# B&R Automation Studio project stroj
Automation Studio 4.10.2.37; technology packages: mapp 5.14.1, mappView 5.14.2

## Configuration Config1

CPU 4PPC30.0702-22B, AutomationRuntime B4.91, Build 4.1.2, Vc V4.72.3

CPU 4PPC30.0702-23B, AutomationRuntime B4.91, Build 4.1.2, Vc V4.72.3

### Task classes (Cpu.sw)
```
Cyclic#1 (cycle 10000 us, tolerance 10000 us):
  TempReg <- TempReg.prg
Cyclic#3 (cycle 50000 us, tolerance 50000 us):
  Machine_Co <- Machine_Control.prg
  Recipes <- Recipes.prg
  VizControl <- Visualization.VizControls.prg
VcDataObjects: Visu <- Visualization.Visu.dob
Binaries: mvLoader, FWRules, arsvcreg, udbdef, TCData, vcnet, vcrt, vccnum, vctcal, vcdsint, Visu03, vcfile, vcgclass, vccstr, vcpdsw, vccshape, arial, vccbmp, vcmgr, vcshared, vcdsloc, vcctext, Visu02, vccovl, vcfntttf, arialbd, vcalarm, vcpdvnc, vcpfar00, vccbtn, Visu01, vcbclass, vcclbox, arconfig, User, Role, Config, iomap, asfw, ashwac, ashwd, sysconf
Libraries: standard, MpRecipe, MpBase, sys_lib, runtime, MpFile, FileIO, astime, arssl, asieccon, vcresman, asbrstr, asusb, dataobj
```

### Task classes (Cpu.sw)
```
Cyclic#3 (cycle 50000 us, tolerance 50000 us):
  Machine_Co <- Machine_Control.prg
Cyclic#4 (cycle 100000 us, tolerance 100000 us):
  Recipes <- Recipes.prg
  VizControl <- VizControls.prg
VcDataObjects: Visu <- Visualization.Visu.dob
Binaries: mvLoader, FWRules, arsvcreg, udbdef, TCData, arconfig, User, Role, Config, iomap, asfw, ashwac, ashwd, sysconf
Libraries: standard, MpRecipe, MpBase, sys_lib, runtime, astime, arssl, asieccon, MpFile, FileIO
```

### Hardware
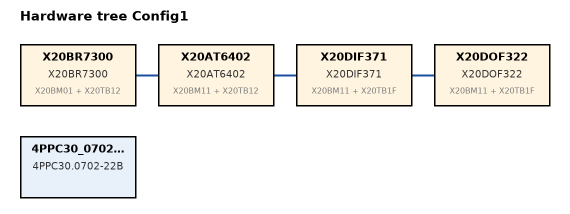
```
4PPC30_0702_22B : 4PPC30.0702-22B v1.1.3.0
  Connector IF3:
    ActivateDevice = 1
    Mode = Manual
    InternetAddress = 192.168.0.1
    SubnetMask = 255.255.255.0
    Vnc1
    VncKeyMappingFile1 = VC\PS2-Keyboard1.dis
    VncAuthentication1 = 1
    VncPasswordViewOnly1 = v
    VncPasswordViewControl1 = c
    VncMaxConnections1 = 4
    ActivateSnmp = 2
  Connector IF4:
    DeviceParam = /IF=2
    TerminatingResistor = 1
  Connector IF8:
    DeviceParam = /CLK=1843200 /CARD=68 /IF=1
  ConfigurationID = stroj_Config1
  EnableUsbRemoteInstall = 1
  TimerDeviceType = SWIOTIMER
  Cyclic1Duration = 10000
  Cyclic1Tolerance = 10000
  Cyclic2Duration = 20000
  Cyclic2Tolerance = 20000
  Cyclic3Duration = 50000
  Cyclic3Tolerance = 50000
  Cyclic4Duration = 100000
  Cyclic4Tolerance = 100000
  Cyclic5Duration = 200000
  Cyclic5Tolerance = 200000
  Cyclic6Duration = 500000
  Cyclic6Tolerance = 500000
  Cyclic7Duration = 1000000
  Cyclic7Tolerance = 1000000
  Cyclic8Duration = 10000
  Cyclic8Tolerance = 30000000
  FileDevice1
  FileDeviceName1 = Recipe
  FileDevicePath1 = C:\Projects\Recipes
  ActivateDtmServer = 1
  VcObjectName = Visu
  RotationAngle = 180
  KeyMappingFile = VC\4PPC30_0702_22B.dis
X20AT6402 : X20AT6402 v1.1.0.0  [SS1 -> X20TB12a.SS; SL -> X20BM11.SL1]
  FunctionModel = CANIOBusController
X20BM01 : X20BM01 v2.1.0.0
X20BM11 : X20BM11 v1.0.0.1  [X2X1 -> X20BM01.IF1]
X20BM11a : X20BM11 v1.0.0.1  [X2X1 -> X20BM11.X2X2]
X20BM11b : X20BM11 v1.0.0.1  [X2X1 -> X20BM11a.X2X2]
X20BR7300 : X20BR7300 v1.4.0.0  [CAN1 -> 4PPC30_0702_22B.IF4; SL -> X20BM01.SL1; SS1 -> X20TB12.SS]
  Supervision = off
X20DIF371 : X20DIF371 v1.1.0.0  [SS1 -> X20TB1F.SS; SL -> X20BM11a.SL1]
  FunctionModel = CANIOBusController
X20DOF322 : X20DOF322 v1.4.0.0  [SS1 -> X20TB1F1.SS; SL -> X20BM11b.SL1]
  FunctionModel = CANIOBusController
X20TB12 : X20TB12 v1.0.0.0
X20TB12a : X20TB12 v1.0.0.0
X20TB1F : X20TB1F v1.0.0.0
X20TB1F1 : X20TB1F v1.0.0.0
```

### IoMap.iom - 4PPC30_0702_23B/IoMap.iom
```iecst
VAR_CONFIG
	::gDoHeatingZone1 AT %QX."X20DOF322".DigitalOutput05; (*24 VDC / 0.5 A, source (Heat zone 1)*)
	::gDoHeatingZone2 AT %QX."X20DOF322".DigitalOutput07; (*24 VDC / 0.5 A, source (Heat zone 2)*)
	::gDoHeatingZone3 AT %QX."X20DOF322".DigitalOutput11; (*24 VDC / 0.5 A, source (Heat zone 3)*)
	::gCurrentTemperatures.temperatureHeatZone1 AT %IW."X20AT6402".Temperature01;
	::gCurrentTemperatures.temperatureHeatZone2 AT %IW."X20AT6402".Temperature02;
	::gCurrentTemperatures.temperatureHeatZone3 AT %IW."X20AT6402".Temperature03;
	::gCurrentTemperatures.temperatureIRSensor AT %IW."X20AT6402".Temperature05;
	::gDoVacuum AT %QX."X20DOF322".DigitalOutput02;
	::gDoFreeItem AT %QX."X20DOF322".DigitalOutput04;
	::gDoMaterial AT %QX."X20DOF322".DigitalOutput06;
	::gDoHeating AT %QX."X20DOF322".DigitalOutput08;
	::gDoFrameDown AT %QX."X20DOF322".DigitalOutput10;
	::gDoFrameUp AT %QX."X20DOF322".DigitalOutput12;
	::gDoFormUp AT %QX."X20DOF322".DigitalOutput14;
	::gDoLedControl AT %QX."X20DOF322".DigitalOutput15;
	::gDoCooling AT %QX."X20DOF322".DigitalOutput01;
	::gDoAirPump AT %QX."X20DOF322".DigitalOutput03;
	::gDiSafe_OK AT %IX."X20DIF371".DigitalInput01;
	::gDiQF1_OK AT %IX."X20DIF371".DigitalInput11;
	::gDiQF2_OK AT %IX."X20DIF371".DigitalInput13;
	::gDiQF3_OK AT %IX."X20DIF371".DigitalInput15;
	::gDiButtonStart AT %IX."X20DIF371".DigitalInput03;
	::gDiHeatingLow AT %IX."X20DIF371".DigitalInput02;
	::gDiHeatingHigh AT %IX."X20DIF371".DigitalInput04;
	::gDiFrameUpPoistion AT %IX."X20DIF371".DigitalInput06;
	::gDiFrameDownPosition AT %IX."X20DIF371".DigitalInput08;
	::gDiFormDownPosition AT %IX."X20DIF371".DigitalInput10;
	::gDiFormUpPosition AT %IX."X20DIF371".DigitalInput12;
END_VAR
```

## Configuration Final

CPU 4PPC30.0702-22B, AutomationRuntime B4.91, Build 4.1.2, Vc V4.72.3

### Task classes (Cpu.sw)
```
Cyclic#1 (cycle 10000 us, tolerance 10000 us):
  TempReg <- TempReg.prg
Cyclic#3 (cycle 50000 us, tolerance 50000 us):
  Machine_Co <- Machine_Control.prg
  Recipes <- Recipes.prg
  VizControl <- Visualization.VizControls.prg
VcDataObjects: Visu <- Visualization.Visu.dob
Binaries: udbdef, mvLoader, FWRules, TCData, sysconf, Role, User, iomap, ashwd, asfw, arconfig, ashwac
Libraries: runtime, arssl, fileio
```

### Hardware
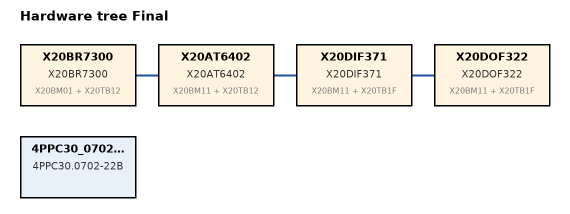
```
4PPC30_0702_22B : 4PPC30.0702-22B v1.1.3.0
  Connector IF3:
    ActivateDevice = 1
  ConfigurationID = stroj_Final
  Simulation = 1
  TimerDeviceType = SWIOTIMER
  Cyclic1Duration = 10000
  Cyclic1Tolerance = 10000
  Cyclic2Duration = 20000
  Cyclic2Tolerance = 20000
  Cyclic3Duration = 50000
  Cyclic3Tolerance = 50000
  Cyclic4Duration = 100000
  Cyclic4Tolerance = 100000
  Cyclic5Duration = 200000
  Cyclic5Tolerance = 200000
  Cyclic6Duration = 500000
  Cyclic6Tolerance = 500000
  Cyclic7Duration = 1000000
  Cyclic7Tolerance = 1000000
  Cyclic8Duration = 10000
  Cyclic8Tolerance = 30000000
  FileDevice1
  FileDeviceName1 = Recipes
  FileDevicePath1 = D:\
  VcObjectName = Visu
  RotationAngle = 180
  KeyMappingFile = VC\4PPC30_0702_22B.dis
X20AT6402 : X20AT6402 v1.1.0.0  [SS1 -> X20TB12.SS; SL -> X20BM11.SL1]
  FunctionModel = CANIOBusController
X20BM01a : X20BM01 v2.1.0.0
X20BM11 : X20BM11 v1.0.0.1  [X2X1 -> X20BM01a.IF1]
X20BM11a : X20BM11 v1.0.0.1  [X2X1 -> X20BM11.X2X2]
X20BM11b : X20BM11 v1.0.0.1  [X2X1 -> X20BM11a.X2X2]
X20BR7300 : X20BR7300 v1.4.0.0  [CAN1 -> 4PPC30_0702_22B.IF4 (NodeNumber=1); SL -> X20BM01a.SL1; SS1 -> X20TB12a.SS]
X20DIF371 : X20DIF371 v1.1.0.0  [SS1 -> X20TB1F.SS; SL -> X20BM11a.SL1]
  FunctionModel = CANIOBusController
X20DOF322 : X20DOF322 v1.4.0.0  [SS1 -> X20TB1F1.SS; SL -> X20BM11b.SL1]
  FunctionModel = CANIOBusController
X20TB12 : X20TB12 v1.0.0.0
X20TB12a : X20TB12 v1.0.0.0
X20TB1F : X20TB1F v1.0.0.0
X20TB1F1 : X20TB1F v1.0.0.0
```

### IoMap.iom - 4PPC30_0702_22B/IoMap.iom
```iecst
VAR_CONFIG
	::gDiSafe_OK AT %IX."X20DIF371".DigitalInput01;
	::gDiHeatingBack AT %IX."X20DIF371".DigitalInput02;
	::gDiQF1_OK AT %IX."X20DIF371".DigitalInput11 INVERSE;
	::gDiQF2_OK AT %IX."X20DIF371".DigitalInput13 INVERSE;
	::gDiQF3_OK AT %IX."X20DIF371".DigitalInput15 INVERSE;
	::gDiHeatingFront AT %IX."X20DIF371".DigitalInput04;
	::gDiFrameUpPoistion AT %IX."X20DIF371".DigitalInput06;
	::gDiFrameDownPosition AT %IX."X20DIF371".DigitalInput08;
	::gDiFormDownPosition AT %IX."X20DIF371".DigitalInput10;
	::gDiButtonStart AT %IX."X20DIF371".DigitalInput03;
	::gDoCooling AT %QX."X20DOF322".DigitalOutput01;
	::gDoHeatingZone1 AT %QX."X20DOF322".DigitalOutput05;
	::gDoHeatingZone2 AT %QX."X20DOF322".DigitalOutput07;
	::gDoLedControl AT %QX."X20DOF322".DigitalOutput15;
	::gDoVacuum AT %QX."X20DOF322".DigitalOutput02;
	::gDoAirPump AT %QX."X20DOF322".DigitalOutput03;
	::gDoFreeItem AT %QX."X20DOF322".DigitalOutput04;
	::gDoMaterial AT %QX."X20DOF322".DigitalOutput06;
	::gDoHeating AT %QX."X20DOF322".DigitalOutput08;
	::gDoFrameDown AT %QX."X20DOF322".DigitalOutput10;
	::gDoFrameUp AT %QX."X20DOF322".DigitalOutput12;
	::gDoFormUp AT %QX."X20DOF322".DigitalOutput14;
	::gCurrentTemperatures.temperatureHeatZone1 AT %IW."X20AT6402".Temperature01;
	::gCurrentTemperatures.temperatureHeatZone2 AT %IW."X20AT6402".Temperature02;
	::gCurrentTemperatures.temperatureHeatZone3 AT %IW."X20AT6402".Temperature03;
	::gCurrentTemperatures.temperatureIRSensor AT %IW."X20AT6402".Temperature05;
	::gDiFormUpPosition AT %IX."X20DIF371".DigitalInput12;
	::gDoHeatingZone3 AT %QX."X20DOF322".DigitalOutput09;
END_VAR
```

## Logical view

Binary libraries used (declarations not repeated): operator, runtime, astime, AsIecCon, standard, MpRecipe, MpBase, sys_lib

### Global.typ - Global data types
```iecst
TYPE
	StateOfProcessType :
		(
		ManualMode,
		DefaultState,
		Start,
		BubbleANDFormDownDelay,
		StartForming,
		CoolingANDBlowingDelay,
		Finishing
		);
	TemperaturesType : 	STRUCT
		temperatureHeatZone1 : INT;
		temperatureHeatZone2 : INT;
		temperatureHeatZone3 : INT;
		temperatureIRSensor : INT;
		temperatureOffset : INT;
		temperatureHysterese : REAL;
	END_STRUCT;
	TimersType : 	STRUCT
		HeatingTOFValue : REAL;
		BlowingTONValue : REAL;
		BlowingTOFValue : REAL;
		BubbleTOFValue : REAL;
		FormingTONValue : REAL;
		FormLockingTONValue : REAL;
		FormingTOFVALUE : REAL;
		FreeItemTOFValue : REAL;
		FreeItemTONValue : REAL;
		FormUpTONValue : REAL;
	END_STRUCT;
END_TYPE
```

### Global.var - Global variables
```iecst
VAR
	gDoMaterial : BOOL;
	gDiButtonStart : BOOL;
	gDiQF2_OK : BOOL;
	gDoCooling : BOOL;
	gDoAirPump : BOOL;
	gDiSafe_OK : BOOL;
	gDiQF1_OK : BOOL;
	gDiFrameUpPoistion : BOOL;
	gDiHeatingLow : BOOL;
	gDiHeatingHigh : BOOL;
	gDoFormUp : BOOL;
	gDiQF3_OK : BOOL;
	gDoLedControl : BOOL;
	gDoHeatingZone2 : BOOL;
	gDiFrameDownPosition : BOOL;
	gDoHeatingZone1 : BOOL;
	gDoVacuum : BOOL;
	gDoFreeItem : BOOL;
	gDoHeatingZone3 : BOOL;
	gDoFrameDown : BOOL;
	gDoFrameUp : BOOL;
	gDiFormDownPosition : BOOL;
	gDiFormUpPosition : BOOL;
	gDoHeating : BOOL;
	gAiIRSensor : INT;
	gAiHeatingZone1 : INT;
	gAiHeatingZone3 : INT;
	gAiHeatingZone2 : INT;
	gAVGTemperature : INT;
	gStateOfProcess : StateOfProcessType;
	gSetTemperatures : TemperaturesType;
	gSetTimersValues : TimersType;
	gRecipeLoaded : BOOL;
	gCurrentTemperatures : TemperaturesType;
	gDiHeatingFront : BOOL;
	gDiHeatingBack : BOOL;
	gHeatingZone1Ready : BOOL;
	gHeatingZone2Ready : BOOL;
	gHeatingZone3Ready : BOOL;
END_VAR
```


### Program Logical/Machine_Control (IEC)

#### Main.st - Init, cyclic, exit code
```iecst
PROGRAM _INIT
	//Start state of cyclus
	gStateOfProcess := ManualMode;
	//--------------------------------------------------------------------------------------------
END_PROGRAM

PROGRAM _CYCLIC
	ManualModeControl;
(*	CASE gStateOfProcess OF
		ManualMode:
			ManualModeControl;

		IF (gDiButtonStart = TRUE) AND (gRecipeLoaded = TRUE) THEN
			cmdAirPump := gDiButtonStart;
			cmdFrameDown := gDiButtonStart;
			IF (gDiFrameDownPosition = TRUE) THEN
				//cmdAirPump:= TRUE/FALSE; ??
				//cmdFrameDown:=TRUE/FALSE; ??
				gStateOfProcess := Start;
			END_IF;
		END_IF;

		Start:
			cmdHeating := TRUE;
			//cmdFrameDown :=TRUE / FALSE;
			//cmdAirPump := TRUE  / FALSE;
			TOFHeating.IN := EDGEPOS(cmdHeating);
			TOFHeating.PT := REAL_TO_TIME(gSetTimersValues.HeatingTOFValue * 1000);
			TOFHeating();

			cmdHeating := TOFHeating.Q; //IF gDiHeatingHigh cmdHeating := FALSE ??

			IF (gDiHeatingHigh = TRUE) THEN
				cmdMaterial := TRUE; // kedy vypnuť
				IF (gSetTimersValues.BlowingTONValue <> 0.0) THEN
					TONBlowing.IN := TRUE;
					TONBlowing.PT := REAL_TO_TIME(gSetTimersValues.BlowingTONValue * 1000);
					TONBlowing();

					TOFBlowing.IN := EDGEPOS(TONBlowing.Q);
					TOFBlowing.PT := REAL_TO_TIME(gSetTimersValues.BlowingTONValue * 1000);
					TOFBlowing();
					cmdBlowing := TOFBlowing.Q;

					IF (cmdHeating = FALSE) AND (TOFBlowing.ET = TOFBlowing.PT) THEN
						cmdMaterial := FALSE;
						gStateOfProcess := BubbleANDFormDownDelay;
					END_IF;
				ELSE
					IF (cmdHeating = FALSE) THEN
						cmdMaterial := FALSE;
						gStateOfProcess := BubbleANDFormDownDelay;
					END_IF
				END_IF;

			END_IF;

		BubbleANDFormDownDelay :
			//------------Zpoždení uzavření formy nastavené na x sekund ---------------
			TONFormLocking.IN := TRUE;
			TONFormLocking.PT := REAL_TO_TIME(gSetTimersValues.FormLockingTONValue * 1000);
			TONFormLocking();
			cmdFormUp:= NOT(TONFormLocking.Q); // cmdFormUp ??
			//---------------------------------------------
			//------------Zpoždení formovaní nastastavené na x sekund -----------------------
			TONForming.IN := TONFormLocking.Q;
			TONForming.PT := REAL_TO_TIME(gSetTimersValues.FormingTONValue * 1000);
			TONForming();
			//---------------------------------------------------------------
			//Ovladanie bubliny
			IF (gDiHeatingLow = TRUE) THEN
				IF gSetTimersValues.BubbleTOFValue <> 0 THEN
					//Zapni bublinu na x sekund
					cmdBubble := TRUE;
					TOFBubble.IN := EDGEPOS(cmdBubble);
					TOFBubble.PT := REAL_TO_TIME(gSetTimersValues.BubbleTOFValue * 1000);
					TOFBubble();
					cmdBubble := TOFBubble.Q;
				END_IF;
			END_IF;
			//AK je forma dole vypni bublinu
			IF (gDiFormDownPosition = TRUE) THEN
				cmdBubble := FALSE;
				//--------------------------------------------------
			END_IF;
			//Ak môžme začať formovať a bublina je vypnuta prejdi na krok formovanie
			IF (cmdFormUp = FALSE) AND (cmdBubble = FALSE) AND (gDiFormDownPosition = TRUE) THEN
				gStateOfProcess := StartForming;
			END_IF;
			//--------------------------------------------------
		StartForming :
			//Formovanie na x sekund
			cmdForming := TRUE;
			TOFForming.IN := EDGEPOS(cmdForming);
			TOFForming.PT := REAL_TO_TIME(gSetTimersValues.FormingTOFVALUE * 1000);
			TOFForming();
			cmdForming:=TOFForming.Q; //asi vacuum
			//--------------
			//Ak to skončí formovanie prejdi na ďalší krok
			IF (cmdForming = FALSE) THEN
				gStateOfProcess :=CoolingANDBlowingDelay;
			END_IF;
		CoolingANDBlowingDelay:
			//Zapni chladnie
			//Zapni oneskorenie odfuku na x sekund
			cmdCooling := TRUE;
			TONFreeItem.IN := TRUE;
			TONFreeItem.PT := REAL_TO_TIME(gSetTimersValues.FreeItemTONValue * 1000);
			TONFreeItem();
			//Ak vyprí čas oneskorenia prejdi na ďaľší krok
			IF (TONFreeItem.Q = TRUE) THEN
				gStateOfProcess := Finishing;
			END_IF;
		Finishing:
			//Zapni odfuk na x sekund
			cmdFreeItem:= TRUE;
			TOFFreeItem.IN := cmdFreeItem;
			TOFFreeItem.PT := REAL_TO_TIME(gSetTimersValues.FreeItemTOFValue * 1000);
			TOFFreeItem();
			cmdFreeItem := TOFFreeItem.Q;
			//------------
			//Oneskorenie otvorenia formy nastavené na x sekund
			TONFormUp.IN := TRUE;
			TONFormUp.PT := REAL_TO_TIME(gSetTimersValues.FormUpTONValue);
			TONFormUp();
			IF TONFormUp.Q THEN
				cmdFormUp:=TRUE; //cmdFormUp
				cmdCooling:=FALSE;
				cmdFrameDown := FALSE;
				cmdFrameUp := TRUE;
			END_IF;
			IF (gDiFrameUpPoistion = TRUE) THEN
				cmdFrameUp := FALSE;
				gStateOfProcess := DefaultState;
			END_IF;

	END_CASE;

	*)

END_PROGRAM

PROGRAM _EXIT
END_PROGRAM
```

#### Variables.var - Local variables
```iecst
VAR
	cmdFormUp : BOOL;
	cmdFrameDown : BOOL;
	cmdMaterial : BOOL;
	cmdCooling : BOOL;
	cmdFreeItem : BOOL;
	cmdVacuum : BOOL;
	cmdAirPump : BOOL;
	cmdHeating : BOOL;
	cmdFrameUp : BOOL;
	TOFBubble : TOF;
	TOFBlowing : TOF;
	TOFHeating : TOF;
	TONForming : TON;
	TONBlowing : TON;
	TONFormLocking : TON;
	cmdBlowing : BOOL;
	cmdForming : BOOL;
	cmdBubble : BOOL;
	TOFForming : TOF;
	TONFreeItem : TON;
	TOFFreeItem : TOF;
	TONFormUp : TON;
	cmdHeatingZone1 : BOOL;
	cmdHeatingZone2 : BOOL;
	cmdHeatingZone3 : BOOL;
END_VAR
```

#### ManualModeControl.st
```iecst
ACTION ManualModeControl:
	IF gDiFrameDownPosition = TRUE THEN
		cmdHeating;
		gDoHeating := cmdHeating;
	ELSIF gDiFrameUpPoistion = TRUE THEN
		cmdHeating := FALSE;
		gDoHeating := cmdHeating;
	END_IF;

	IF gDiHeatingBack = TRUE THEN //topení vzadu
		cmdFormUp;
		cmdFrameDown;
		cmdFrameUp;
		gDoFormUp := cmdFormUp;
		gDoFrameDown := cmdFrameDown;
		gDoFrameUp := cmdFrameUp;
	ELSIF gDiHeatingFront = TRUE THEN
		cmdFormUp := FALSE;
		cmdFrameDown := FALSE;
		cmdFrameUp := FALSE;
	END_IF;
	IF (gDiFrameDownPosition = TRUE) AND (gDiFormUpPosition = TRUE) THEN
		cmdHeating := FALSE;
		gDoHeating := cmdHeating;
	END_IF;

	gDoFreeItem := cmdFreeItem;
	gDoMaterial := cmdMaterial;
	gDoAirPump := cmdAirPump;
	gDoCooling := cmdCooling;
	gDoHeatingZone1 := cmdHeatingZone1;
	gDoHeatingZone2 := cmdHeatingZone2;
	gDoHeatingZone3 := cmdHeatingZone3;
	IF gDoAirPump = TRUE THEN
		gDoVacuum := cmdVacuum;
	END_IF
END_ACTION
```

### Program Logical/Recipes (IEC)

#### Variables.var
```iecst
VAR
	MpRecipeXml_0 : MpRecipeXml;
	MpRecipeRegParTemperatures : MpRecipeRegPar;
	MpRecipeRegParTimers : MpRecipeRegPar;
	cmdLoadRecipes : BOOL;
	cmdSaveRecipes : BOOL;
	cmdErrorReset : BOOL;
	RecipeUI : MpRecipeUI;
	UISetup : MpRecipeUISetupType;
	UIConnect : MpRecipeUIConnectType;
END_VAR
```

#### Main.st
```iecst
PROGRAM _INIT
	(* Insert code here *)

	UISetup.RecipeListSize := 5;

END_PROGRAM

PROGRAM _CYCLIC
	(* Insert code here *)

	gDoHeatingZone1;
	MpRecipeXml_0.MpLink := ADR(gRecipeXml);
	MpRecipeXml_0.Enable := TRUE;
	MpRecipeXml_0.DeviceName := ADR('Recipe');
	gRecipeLoaded := UDINT_TO_BOOL(MpRecipeXml_0.Info.FileSize); // check if Recipe is loaded (If not lenght = 0)

	MpRecipeRegParTemperatures.MpLink := ADR(gRecipeXml);
	MpRecipeRegParTemperatures.Enable := MpRecipeXml_0.Active;
	MpRecipeRegParTemperatures.ErrorReset := cmdErrorReset;
	MpRecipeRegParTemperatures.Category := ADR('Temperatures');
	MpRecipeRegParTemperatures.PVName := ADR('gSetTemperatures');

	MpRecipeRegParTimers.MpLink := ADR(gRecipeXml);
	MpRecipeRegParTimers.Enable := MpRecipeXml_0.Active;
	MpRecipeRegParTimers.ErrorReset := cmdErrorReset;
	MpRecipeRegParTimers.Category := ADR('Timers');
	MpRecipeRegParTimers.PVName := ADR('gSetTimersValues');

	RecipeUI.Enable := TRUE;
	RecipeUI.MpLink := ADR(gRecipeXml);
	RecipeUI.UISetup :=UISetup;
	RecipeUI.UIConnect := ADR(UIConnect);

	MpRecipeXml_0();
	MpRecipeRegParTemperatures();
	MpRecipeRegParTimers();
	RecipeUI();
END_PROGRAM

PROGRAM _EXIT
	(* Insert code here *)

END_PROGRAM
```

- Visualisation Logical/Visualization (not shown)

### Program Logical/TempReg (IEC)

#### Variables.var
```iecst
VAR
	HeatZone1HystUpperLimit : REAL;
	HeatZone2HystUpperLimit : REAL;
	HeatZone1HystDownLimit : REAL;
	HeatZone2HystDownLimit : REAL;
	HeatZone3HystDownLimit : REAL;
	HeatZone3HystUpperLimit : REAL;
END_VAR
```

#### Main.st
```iecst
PROGRAM _INIT
	(* Insert code here *)

END_PROGRAM

PROGRAM _CYCLIC
	(* Insert code here *)

END_PROGRAM

PROGRAM _EXIT
	(* Insert code here *)

END_PROGRAM
```

### TurnOfHeating.st - not listed in the package file held
```iecst
ACTION TurnOffHeating:
	gDoHeatingZone1 := FALSE;
	gDoHeatingZone2 := FALSE;
	gDoHeatingZone21 := FALSE;
	gDoHeatingZone3 := FALSE;
	gDoHeatingZone31 :=FALSE;
END_ACTION
```

### TurnOnHeating.st - not listed in the package file held
```iecst
ACTION TurnOnHeating:
	gDoHeatingZone1 := TRUE;
	gDoHeatingZone2 := TRUE;
	gDoHeatingZone21 := TRUE;
	gDoHeatingZone3 := TRUE;
	gDoHeatingZone31 :=TRUE;
END_ACTION
```

### Program Logical/VizControls

#### Variables.var
```iecst
VAR
	ItemIconIndex : USINT;
	MaterialIconIndex : USINT;
	VacuumIconIndex : USINT;
	CoolingIconIndex : USINT;
	HeatingZonesIconIndex : USINT;
	AirPumpIconIndex : USINT;
	FrameDownIndex : USINT;
	FrameUpIconIndex : USINT;
	FormUpIndex : USINT;
	HeatingOnOfText2 : USINT;
	HeatingOnOfText3 : USINT;
	HeatingOnOfText1 : USINT;
END_VAR
```

#### Main.st
```iecst
PROGRAM _INIT
	(* Insert code here *)

END_PROGRAM

PROGRAM _CYCLIC

	IF gDoCooling THEN
		CoolingIconIndex := 4;
	ELSE
		CoolingIconIndex := 10;
	END_IF

	IF gDoAirPump THEN
		AirPumpIconIndex := 6;
	ELSE
		AirPumpIconIndex :=12;
	END_IF
	IF gDoHeatingZone1 THEN
		HeatingOnOfText1 := 1;
	ELSE
		HeatingOnOfText1 := 0;
	END_IF;
	IF gDoHeatingZone2 THEN
		HeatingOnOfText2 := 1;
	ELSE
		HeatingOnOfText2 := 0;
	END_IF;
	IF gDoHeatingZone3 THEN
		HeatingOnOfText3 := 1;
	ELSE
		HeatingOnOfText3 := 0;
	END_IF;
	IF gDoHeatingZone1 AND gDoHeatingZone2 AND gDoHeatingZone3 THEN
		HeatingZonesIconIndex := 7;
	ELSE
		HeatingZonesIconIndex := 13;
	END_IF

	IF gDoVacuum THEN
		VacuumIconIndex := 3;
	ELSE
		VacuumIconIndex := 9;
	END_IF

	IF gDoFreeItem THEN
		ItemIconIndex := 18;
	ELSE
		ItemIconIndex := 21;
	END_IF
	IF gDoFreeItem THEN
		ItemIconIndex := 18;
	ELSE
		ItemIconIndex := 21;
	END_IF

	IF gDoFormUp THEN
		FormUpIndex := 8;
	ELSE
		FormUpIndex := 14;
	END_IF

	IF gDoFrameDown THEN
		FrameDownIndex := 15;
	ELSE
		FrameDownIndex :=11;
	END_IF;

	IF gDoFrameUp THEN
		FrameUpIconIndex := 17;
	ELSE
		FrameUpIconIndex := 16;
	END_IF;

	IF gDoMaterial THEN
		MaterialIconIndex := 19;
	ELSE
		MaterialIconIndex := 20;
	END_IF;

END_PROGRAM

PROGRAM _EXIT
	(* Insert code here *)

END_PROGRAM
```

Listed in the project but not available here: Logical/Machine_Control/Types.typ
